{attribute 'GeneratedUsingTerminal: EL2878-0005-0016'}
{attribute addProperty BoxType "EL2878-0005-0016"}
{attribute addProperty Id "DiagAT %I*BOOL1"}
{attribute addProperty CRC "2804620823"}
{attribute addProperty Size "1"}
TYPE Diagnostic_A72B1E17 :
STRUCT
	{attribute addProperty Name "Diag"}
	Diag AT %I* : BOOL;
END_STRUCT
END_TYPE

(* stored: Version 1.2.0.0, ProductVersion 3.1.4024.9
   DUT Diagnostic_A72B1E17: Id {b373b107-bf68-49c4-9e37-25358a266e78} *)
